(* PLC project Generated.project, CODESYS CODESYS V3.5 SP19 Patch 1 *)
(* stored: creationDateTime 2026-08-11T14:02:33.674168, modificationDateTime 2026-08-11T14:02:33.674168 *)

(* ═══════════════════════════════════════════════════════════════ 🌐 ST_CommunHMI — Données d'échange IHM COMMUNES (pas propres à un axe) ─────────────────────────────────────────────────────────────── 🆕 REX 2026-07-08 (demande utilisateur) : regroupe les signaux qui ne concernent PAS un axe/mécanisme en particulier (1 seul capteur/signal partagé par toute la machine) — évite de les dupliquer ou de les laisser en variables isolées directement dans GVL_IHM. Exemple : TopPositionSensorActive (capteur unique, commun M1+M2), BrakeThermalFault (retour unique, commun M1+M2+M3). ⚠️ Ne pas y mettre HmiInitDone (indicateur interne de séquencement boot, pas une information machine destinée à l'opérateur) — reste seul dans GVL_IHM. ═══════════════════════════════════════════════════════════════ *)
TYPE ST_CommunHMI : STRUCT
  TopPositionSensorActive : BOOL;  (* ⚠️ Capteur de position haute commun M1+M2 détecté *)
  BrakeThermalFault : BOOL;  (* 🌡️ Défaut/perte thermique frein — retour unique commun M1/M2/M3, escalade PowerCutOff *)
  PhaseRotationFault : BOOL;  (* 🆕 REX 2026-07-08 : rotation de phase incorrecte — retour unique commun M1/M2/M3 *)
  LimitLegalReached : BOOL;  (* 📐 Limite légale de profondeur de dragage atteinte (globale) *)
  Cfg : ST_CommunCfg;  (* 🔧 Configuration des paramètres communs machine *)
  HydraulicThermalFault : BOOL;  (* 🆕 REX 2026-07-18 : défaut/perte thermique centrale hydraulique *)
  Bypass : ST_BypassCommun;  (* 🔧 Bypass maintenance de capteurs COMMUNS (voir REGISTRE_ACTIONS_Bypass_v1.0 (archive)) 🆕 2026-08-07 : granulaire, applique le bypass aux 2 treuils simultanement (pilotage "both") — OR avec le bypass individuel M1/M2 dans PRG_04 *)
  SimTopSensorBypassActive : BOOL;  (* 🩺 2026-08-07 : indicateurs diagnostic simulation — PLC→IHM, PAS des bypass operateur (etaient ecrits par erreur dans Bypass.SlackCable/TopPositionSensor avant ce lot, ce qui empechait ces champs de servir de vrai bypass RETAIN operateur). 🩺 Capteur haut ignore car simulation active *)
  SimSlackCableBypassActive : BOOL;  (* 🩺 Mou de cable ignore car simulation active *)
  TglHeartbeatIhm : BOOL;  (* 💓 Heartbeat IHM↔PLC — IHM inverse TglHeartbeatIhm toutes les 500 ms. IHM→PLC : toggle périodique, jamais valeur constante *)
  TglHeartbeatPlc : BOOL;  (* PLC→IHM : clignotant activité PLC *)
  HeartbeatIhmOk : BOOL;  (* PLC→IHM : front IHM post-boot reçu et timeout absent *)
  HeartbeatIhmTimeout : BOOL;  (* PLC→IHM : aucun front IHM depuis 2 s *)
  HeartbeatIhmElapsed : TIME;  (* PLC→IHM : temps depuis dernier front IHM *)
  BtnWinchBothUp : BOOL;  (* 🆕 Boutons pilotage direct des 2 treuils (communs, remplace SelJoystickWinch en mode boutons) ⬆️ Monte les 2 treuils simultanément *)
  BtnWinchBothDown : BOOL;  (* ⬇️ Descend les 2 treuils simultanément *)
  ConfigRestoredFromPersistent : BOOL;  (* 🐛 FIX 2026-07-23 : alarme restauration config PERSISTENT (RETAIN invalidé, ex. changement de struct ST_*HMI) — visible et acquittable, jamais de disparition automatique silencieuse (doctrine reset=front, PRG_SUPERVISION_CFC.st §2bis). Vérifier les valeurs avant reprise cycle. ⚠️ PLC→IHM : restauration détectée ce boot, à vérifier *)
  BtnAckConfigRestored : BOOL;  (* 🔘 IHM→PLC : acquittement opérateur (front) *)
  Preflight : ST_PreflightHMI;  (* 🩺 Verdict observateur à l'arrêt — jamais bloquant *)
  WinchSymmetry : ST_WinchSymmetryHMI;  (* ⚖️ MES-008 : mesures passives M1/M2 *)
  KoboldImmersionConfirmed : BOOL;  (* 🩺 2026-08-07 (Fiche 05) : diagnostic arrêt auto descente Kobold (pilotage normal) Front Kobold confirmé dans la fenêtre d'immersion *)
  KoboldBottomTouchLatched : BOOL;  (* Fond détecté, descente bloquée (ForbidDescentM1/M2_Raw) *)
END_STRUCT;
END_TYPE

(* ═══════════════════════════════════════════════════════════════ 🔧 ST_BypassCommun — Bypass maintenance GRANULAIRE, applicable aux 2 treuils à la fois ─────────────────────────────────────────────────────────────── 🎨 2026-08-07 (demande client) : distinct des bypass individuels M1/M2 (ST_BypassWinch) — un OUI ici lève la protection sur LES DEUX treuils simultanément (pilotage "both", GVL_IHM.Commun.BtnWinchBothUp/Down), en OR avec le bypass individuel de chaque instance (PRG_04_Treuils_Benne). Évite de devoir activer 2 fois le même bypass (M1 ET M2) avant un pilotage groupé — SANS retirer les bypass individuels pour le pilotage à l'unité. ⚠️ Ne remplace PAS les bypass individuels : les deux se combinent en OR, jamais l'un n'entraîne la désactivation de l'autre. 🔒 Doctrine : actionnable UNIQUEMENT en MAINT_N2, RETAIN, jamais masque les autres défauts du même bloc (voir REGISTRE_ACTIONS_Bypass_v1.0 (archive)). 🔧 2026-08-07 : `TopPositionSensor` renommé `TopLimitSwitch` (cohérence avec ST_BypassWinch) — était de toute façon inutilisé comme bypass réel jusqu'ici (PRG_07_Supervision y écrivait un indicateur simulation par erreur, voir ST_CommunHMI.SimTopSensorBypassActive). ═══════════════════════════════════════════════════════════════ *)
TYPE ST_BypassCommun : STRUCT
  SlackCable : BOOL;  (* ⚠️ Bypass capteur mou de câble — capteur unique M1/M2, OR avec bypass individuel *)
  TopLimitSwitch : BOOL;  (* 🚧 Bypass fin de course physique haute (capteur, bit5), OR avec bypass individuel *)
  TopLimitSoftware : BOOL;  (* 🆕 2026-08-07 : Bypass fin de course logiciel haut (position calculée), OR avec bypass individuel *)
  CableLimitSwitch : BOOL;  (* 🆕 2026-08-07 : Bypass limite basse physique (longueur câble), OR avec bypass individuel *)
  LimitLegal : BOOL;  (* 🆕 2026-08-07 : Bypass limite légale de profondeur, OR avec bypass individuel *)
END_STRUCT;
END_TYPE

(* ═══════════════════════════════════════════════════════════════ 🔧 ST_CommunCfg — Configuration des paramètres communs machine 📄 2026-07-24 : WinchMaxStepDescente/WinchMaxStepAscent/WinchSlowdownDistance_M/ WinchSlowSpeed_Pct rapatriés depuis ST_WinchCfg (étaient partagés M1/M2 par réconciliation ad-hoc dans PRG_SUPERVISION_CFC.st, une seule instance ici l'élimine). ═══════════════════════════════════════════════════════════════ *)
TYPE ST_CommunCfg : STRUCT
  LimitLegalDepthMinAllowed_M : REAL := -999;  (* 🔴🔧 REX 2026-08-07 (5) — retour terrain, blocage instantané à 0m : sans défaut explicite, ce champ vaut 0.0 tant qu'il n'a pas été réglé côté IHM -- "CablePosM <= 0.0" se déclenche dès la position de référence, avant tout réglage réel de la cote légale. Défaut -999.0 (jamais atteint en pratique) : LimitLegalEnabled=TRUE sans réglage ne bloque plus rien par erreur -- il faut régler la vraie cote pour que la protection devienne active. 📐 Cote min de dragage autorisée (m, négatif) *)
  LimitLegalEnabled : BOOL;  (* 🟢 Activation de la limite légale *)
  SelHomingApproachEnable : BOOL;  (* 🔌 Case IHM : autorise le dépassement butée haute pour homing (si MAINT_N2) *)
  WinchMaxStepDescente : INT := 3;  (* 🛑 Limitation palier vitesse en descente (1..5), commun M1/M2 *)
  WinchMaxStepAscent : INT := 5;  (* 🚀 Limitation palier vitesse en montée (1..5), commun M1/M2 *)
  WinchSlowdownDistance_M : REAL := 1;  (* 📏 Distance avant limite pour enclencher le ralentissement (m), commun M1/M2 *)
  WinchSlowdownMaxStep : INT := 1;  (* 🔧 2026-08-07 : WinchSlowSpeed_Pct (%) retiré — un treuil ne connaît que des paliers (1..5), pas une vitesse continue. 🆕 2026-08-07 : Plafond palier dans la zone de ralentissement (1..5), commun M1/M2 *)
  TglEnableKoboldAutoStopDescent : BOOL := FALSE;  (* 🆕 2026-08-07 : Arrêt auto descente sur détection fond Kobold (pilotage normal) *)
  TglEnableCoupledBucketSequencing : BOOL := FALSE;  (* 🔴🔧 REX 2026-08-07 (4) — coupe-circuit d'urgence pour le séquencement auto benne (Fiche 01). Défaut FALSE = comportement IDENTIQUE à avant Fiche 01 (déplacement M1/M2 synchro jamais gouverné par instBucket.Busy sauf action MANUELLE benne/DumpAtTremie/ExtractionSequence). *)
  Initialized : BOOL := FALSE;  (* 🚦 flag restauration boot *)
END_STRUCT;
END_TYPE

TYPE ST_PreflightHMI : STRUCT
  BtnRun : BOOL;
  PreflightOk : BOOL;
  PreflightDone : BOOL;
  PreflightBusy : BOOL;
  PreflightErrorId : WORD;
END_STRUCT;
END_TYPE

TYPE ST_WinchSymmetryHMI : STRUCT
  BtnReset : BOOL;
  SymmetryOk : BOOL;
  SymmetryValid : BOOL;
  DeltaStartDelay_Ms : UDINT;
  DeltaBrakeReleaseTime_Ms : UDINT;
  DeltaBrakeApplyTime_Ms : UDINT;
  DeltaStopDistance_M : REAL;
  DeltaStopTime_Ms : UDINT;
  MaxSyncDeviation_M : REAL;
END_STRUCT;
END_TYPE
